RoboDK station: GoodBoy.rdk

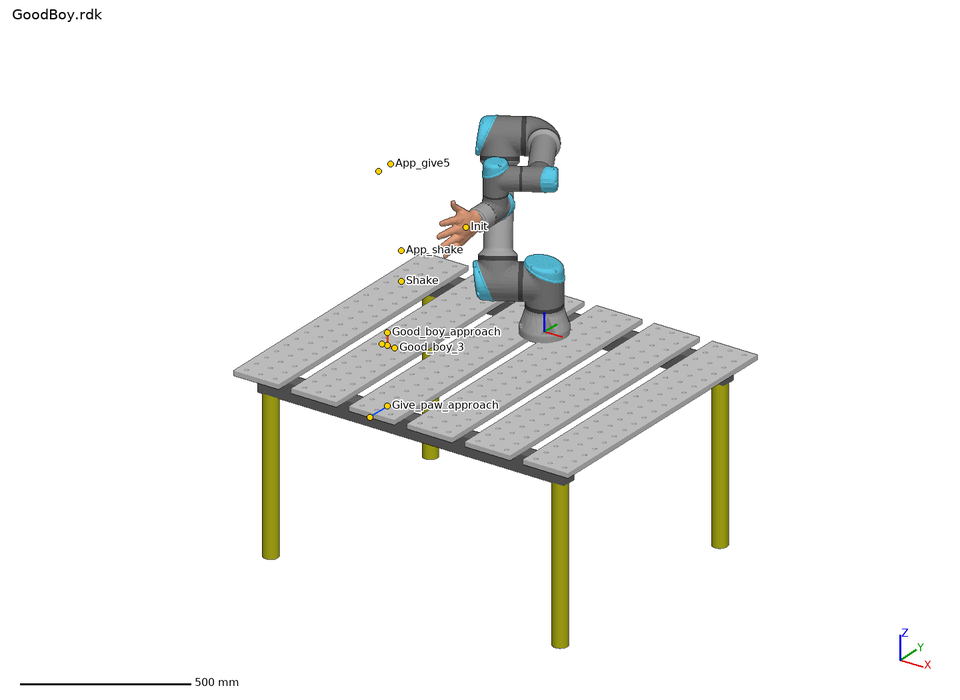
[picture v0: the station drawn from its stored meshes, robots at their saved joint values, targets as dots, program paths as lines]
Station Assistive_UR5e_SW (saved by RoboDK 5.9.2). Poses are relative to the parent item; angles as X-Y-Z fixed-axis rotations.
  - frame UR5e Base at (0, 0, 0) mm
    - robot UR5e: 6 axes, payload 5 kg, reach 850 mm, repeatability 0.03 mm, weight 18.4 kg
        modified DH rows (alpha deg, a mm, theta deg, d mm): 0, 0, 0, 162.5; 90, 0, 180, 0; 0, 425, 0, 0; 0, 392.25, 0, 133.3; -90, 0, 0, 99.7; 90, 0, 180, 99.6
        joint limits [-360, -360, -360, -360, -360, -360] to [360, 360, 360, 360, 360, 360]; home [0, -90, -90, 0, 90, 0]; saved at [-57.836, -65.392, -107.167, 172.559, -57.836, 0]
      - tool Hand, TCP at (0, 0, 50) mm, size 54.8 x 155.9 x 193.5 mm, geometry from Hand.stl
  - frame World at (0, 0, 0) mm
    - object Table at (0, 0, 0) mm, size 1193.8 x 965.2 x 609.6 mm, geometry from welding_table.sld
    - target Init (Cartesian target) at (0, -400, 500) mm, rotated rx 90 ry 0 rz 0 deg; joints [-57.836, -65.392, -107.167, 172.559, -57.836, 0] of UR5e
    - target App_shake (joint target) at (-300, -300, 300) mm, rotated rx 90 ry 0 rz 0 deg; joints [-129.97, -84.968, -123.366, -151.667, -129.97, 0] of UR5e
    - target Shake (joint target) at (-300, -300, 200) mm, rotated rx 90 ry 0 rz 0 deg; joints [-129.97, -95.332, -131.473, -133.195, -129.97, 0] of UR5e
    - target App_give5 (joint target) at (-380.86, -238.62, 533.82) mm, rotated rx 0 ry 0 rz 90 deg; joints [-130.679, -89.195, -122.013, 301.208, -90, 130.679] of UR5e
    - target Give5 (joint target) at (-380.86, -300, 533.82) mm, rotated rx 0 ry 0 rz 90 deg; joints [-125.814, -94.091, -116.939, 301.03, -90, 125.814] of UR5e
    - target Give_paw_approach (Cartesian target) at (0, -798.62, 77.84) mm, rotated rx -90 ry 90 rz -180 deg; joints [-78.148, -141.493, -78.021, 219.514, -78.148, -90.003] of UR5e
    - target Give_paw (Cartesian target) at (0, -887.97, 77.84) mm, rotated rx -90 ry 90 rz -180 deg; joints [-79.599, -152.701, -54.595, 207.296, -79.599, -90.003] of UR5e
    - target Good_boy_approach (Cartesian target) at (0.01, -798.62, 315.42) mm, rotated rx 90 ry -89.25 rz 0 deg; joints [-78.147, -126.553, -66.529, 193.082, -78.147, 89.251] of UR5e
    - target Good_boy_1 (Cartesian target) at (-0.52, -798.62, 274.91) mm, rotated rx 90 ry -89.25 rz 0 deg; joints [-78.193, -128.135, -70.012, 198.147, -78.193, 89.251] of UR5e
    - target Good_boy_2 (Cartesian target) at (-20.77, -798.62, 273.61) mm, rotated rx -90 ry -86.32 rz 180 deg; joints [-79.987, -128.24, -70.034, 198.274, -79.987, 93.683] of UR5e
    - target Good_boy_3 (Cartesian target) at (24.89, -798.62, 273.67) mm, rotated rx 90 ry -87.2 rz 0 deg; joints [-75.961, -128.257, -69.995, 198.253, -75.961, 87.196] of UR5e
  - program Init (3 instructions, listed below)
  - program Give_paw (5 instructions, listed below)
  - program Good_boy (9 instructions, listed below)
  - program MainProgram (4 instructions, listed below)
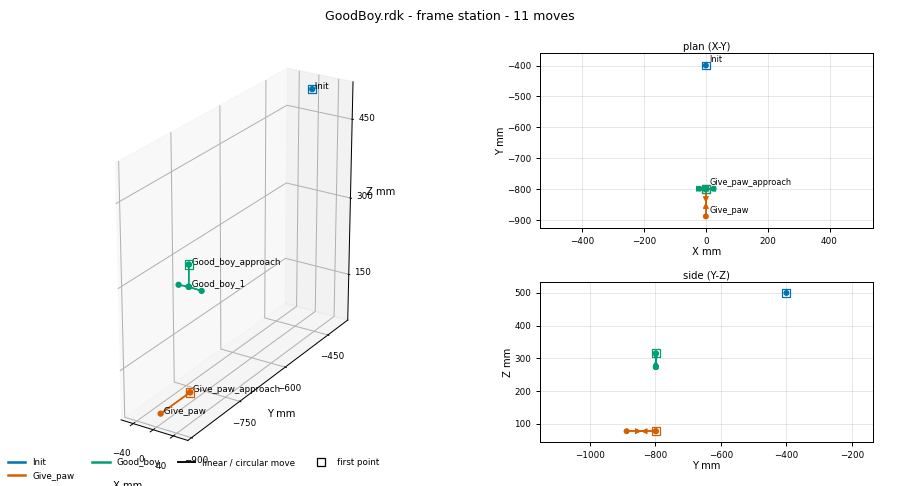
[picture p0: tool path of GoodBoy.rdk in frame station, 11 of 11 moves have a stored position in this frame; points joined in program order, loops and branches not executed]

--- program Init (robot UR5e) ---
  Est. Ref.: UR5e Base
  Est. herr: Hand
  MoveJ (Init)

--- program Give_paw (robot UR5e) ---
  Est. Ref.: UR5e Base
  Est. herr: Hand
  MoveL (Give_paw_approach)
  MoveL (Give_paw)
  MoveL (Give_paw_approach)

--- program Good_boy (robot UR5e) ---
  Est. Ref.: UR5e Base
  Est. herr: Hand
  MoveL (Good_boy_approach)
  MoveL (Good_boy) -> target Good_boy_1
  MoveL (Good_boy_2)
  MoveL (Good_boy_1)
  MoveL (Good_boy_3)
  MoveL (Good_boy_1)
  MoveL (Good_boy_approach)

--- program MainProgram (robot UR5e) ---
  Llamar Init
  Llamar Give_paw
  Llamar Good_boy
  Llamar Init
